FUNCTION_BLOCK ABSTRACT FBA_Drive IMPLEMENTS I_Drive
VAR_INPUT
	bEnable : BOOL;
END_VAR
VAR_OUTPUT
	contactSensor AT %I* : BOOL;
	
	outerLimit AT %I* : BOOL;
	home AT %I* : BOOL;
	innerLimit AT %I* : BOOL;
	(*
	busy : BOOL;
	contact : BOOL;
	error : BOOL;
	homeSet : BOOL;
	*)
	homingComplete : BOOL;
END_VAR
VAR
	step : Homing;
END_VAR
(*
this abstract FB only contains the bare minimum types for any drive/servo
*)

{attribute 'monitoring':='call'}
PROPERTY AtHome : BOOL
GET
AtHome := home;
END_GET
END_PROPERTY

{attribute 'monitoring':='call'}
PROPERTY AtInnerLimit : BOOL
GET
AtInnerLimit := innerLimit;
END_GET
END_PROPERTY

{attribute 'monitoring':='call'}
PROPERTY AtOuterLimit : BOOL
GET
AtOuterLimit := outerLimit;
END_GET
END_PROPERTY

{attribute 'monitoring':='call'}
PROPERTY ABSTRACT Busy : BOOL
GET
END_GET
END_PROPERTY

{attribute 'monitoring':='call'}
PROPERTY Contact : BOOL
GET
Contact := contactSensor;
END_GET
END_PROPERTY

{attribute 'monitoring':='call'}
PROPERTY ABSTRACT Error : BOOL
GET
END_GET
END_PROPERTY

PROPERTY HomeSet : BOOL
GET
HomeSet := homingComplete;
END_GET
END_PROPERTY

METHOD ABSTRACT homingSequence : BOOL
VAR_INPUT
END_VAR
END_METHOD

METHOD ABSTRACT reset : BOOL
VAR_INPUT
END_VAR
END_METHOD

METHOD ABSTRACT stop : BOOL
VAR_INPUT
END_VAR
END_METHOD

END_FUNCTION_BLOCK

(* stored: Version 1.1.0.1, ProductVersion 3.1.4024.11
   POU FBA_Drive: Id {8658c98e-873c-4e2d-a515-69a316227735}, SpecialFunc None
   Folder Abstract: Id {4de43f22-8200-4f92-8cad-2bd0fffc60d8}
   Folder Complete: Id {ea622ce6-4632-480e-8e6c-9f050cd2da6f}
   Property AtHome: Id {f5b76a30-248f-4668-ade8-2b6f6ec2c3e3}
   Get Get: Id {d5adc3f1-7d42-444b-9ed3-c000f26174cf}
   Property AtInnerLimit: Id {b968d47e-33dc-4e0f-b026-4fb76aa61d26}
   Get Get: Id {cd7ff1e2-65b0-4e28-b52f-2460f259be3e}
   Property AtOuterLimit: Id {a5069dbd-3ff8-427c-86ff-c2b4c68678c2}
   Get Get: Id {079bb1f6-5cdc-4453-8a86-cf5ae9532eec}
   Property Busy: Id {61d3d1f4-24a5-4614-a13f-353d54ff6c6f}
   Get Get: Id {bd81f5ef-6461-480c-addc-61aba7e1d1f3}
   Property Contact: Id {8985c792-f8f6-4e8b-b6e0-9e7f1830f526}
   Get Get: Id {fa898aee-162a-4214-8a1f-233e8bf413b7}
   Property Error: Id {89c2e4e9-2d12-4706-892e-07677a2ab27e}
   Get Get: Id {4fbcf804-5ac3-41df-bf23-eda104f47c0d}
   Property HomeSet: Id {996846ee-1b00-41ce-9f66-f1c9a22068ed}
   Get Get: Id {4ac52942-bb06-4b10-b6d5-2a04e1b21de8}
   Method homingSequence: Id {390c2a5c-3fb8-494a-86b1-6eaeba5607f6}
   Method reset: Id {a394f766-1996-4b79-b2df-c401a7e36f4b}
   Method stop: Id {b7d827f0-bac0-4ebc-b575-923998f8293d} *)
